{attribute addProperty BoxType "EL2212-0000-0020"}
{attribute addProperty Id "DOX_Status_ChannelAT %I*ARRAY[0..1] OF DOX_Status_Channel_C7709C9E3240DOX_Control_ChannelAT %Q*ARRAY[0..1] OF DOX_Control_Channel_08FE49103240WcStateAT %I*WcState_98A4DF7520.250InfoDataAT %I*InfoData_BC63D37F80100"}
{attribute addProperty CRC "2865043229"}
{attribute addProperty SizeInBites "146"}
{attribute addProperty SizeInBytes "18.25"}
TYPE EL2212_1A3ABF19 :
STRUCT
	{attribute addProperty Name "DOX_Status_Channel"}
	DOX_Status_Channel : ARRAY[0..1] OF DOX_Status_Channel_C7709C9E;
	{attribute addProperty Name "DOX_Control_Channel"}
	DOX_Control_Channel : ARRAY[0..1] OF DOX_Control_Channel_08FE4910;
	{attribute addProperty Name "WcState"}
	WcState : WcState_98A4DF75;
	{attribute addProperty Name "InfoData"}
	InfoData : InfoData_BC63D37F;
END_STRUCT
END_TYPE

(* stored: Version 1.2.0.0, ProductVersion 3.1.4024.9
   DUT EL2212_1A3ABF19: Id {7cf09301-7e5d-423c-a561-2ed679ef1536} *)
